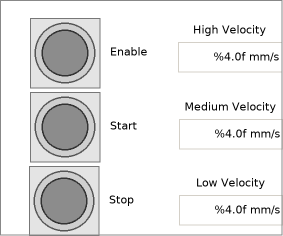
VISUALIZATION Controls  // 283x236
    PushSwitchLed (30,18 70x70), variable: MainCommands.Enable, behaviour: TOGGLE, style: Switch-PushSwitchLed-Gray
    Label (107,37 75x30), "Enable"
    Label (107,111 75x30), "Start"
    PushSwitchLed (30,92 70x70), variable: MainCommands.Start, behaviour: TOGGLE, style: Switch-PushSwitchLed-Gray
    Label (106,185 75x30), "Stop"
    PushSwitchLed (29,166 70x70), variable: MainCommands.Stop, behaviour: TOGGLE, style: Switch-PushSwitchLed-Gray
    Textfield (178,42 104x30), "%4.0f mm/s", text variable: MainCommands.highVelocity
        OnMouseClick: write the text variable via VisuDialogs.Numpad, min 1, max 2000, format %f.0
    Label (181,21 97x18), "High Velocity"
    Textfield (179,119 104x30), "%4.0f mm/s", text variable: MainCommands.mediumVelocity
        OnMouseClick: write the text variable via VisuDialogs.Numpad, min 1, max 2000, format %f.0
    Label (182,98 97x18), "Medium Velocity"
    Textfield (179,195 104x30), "%4.0f mm/s", text variable: MainCommands.lowVelocity
        OnMouseClick: write the text variable via VisuDialogs.Numpad, min 1, max 2000, format %f.0
    Label (182,174 97x18), "Low Velocity"
END_VISUALIZATION

(* stored: Version 1.1.0.1, ProductVersion 3.1.4026.12
   Visu Controls: Id {f1ba0824-aba4-4e43-a127-edb3220c5b1f} *)
